KUKA KRL program: sps.sub

&ACCESS RVEO
&REL 86
&COMMENT PLC on control
DEF  SPS ( )
  ;FOLD DECLARATIONS
  ;FOLD BASISTECH DECL
  ;Automatik extern
  DECL STATE_T STAT
  DECL MODUS_T MODE
  ;ENDFOLD (BASISTECH DECL)
  ;FOLD USER DECL
  ; Please insert user defined declarations

  ;ENDFOLD (USER DECL)
  ;ENDFOLD (DECLARATIONS)
  ;FOLD INI
  ;FOLD DEFAULT MSG_T
  $MSG_T={MSG_T: VALID FALSE,RELEASE FALSE,TYP #NOTIFY,MODUL[] " ",KEY[] " ",PARAM_TYP #VALUE,PARAM[] " ",DLG_FORMAT[] " ",ANSWER 0}
  ;ENDFOLD (DEFAULT MSG_T)
  ;FOLD AUTOEXT INIT
  INTERRUPT DECL 91 WHEN $PRO_STATE1==#P_FREE DO RESET_OUT ()
  INTERRUPT ON 91
  $LOOP_MSG[]="                                                            "
  MODE=#SYNC
  $H_POS=$H_POS
  ;Automatik extern
  IF $MODE_OP==#EX THEN
    CWRITE($CMD,STAT,MODE,"RUN /R1/CELL()")
  ENDIF
  ;ENDFOLD (AUTOEXT INIT)
  ;FOLD USER INIT
  ; Please insert user defined initialization commands
      sws_set = true

  ;ENDFOLD (USER INIT)
  ;ENDFOLD (INI)

  LOOP
     WAIT FOR NOT($POWER_FAIL)

    ;FOLD USER PLC

; Run toolchanger code
toolchanger()
; Update FTC data
updatetoolforces()




    ;ENDFOLD (USER PLC)
  ENDLOOP
  ;FOLD ;%{H}
  ;FOLD
END
  ;ENDFOLD


DEF  RESET_OUT ( )
  INT N
  $LOOP_MSG[]="                                                            "
  IF REFLECT_PROG_NR == 1 THEN
    FOR N = 0 TO PGNO_LENGTH - 1
      $OUT[PGNO_FBIT_REFL + N] = FALSE
    ENDFOR
  ENDIF
  IF (PGNO_REQ>0) THEN
    $OUT[PGNO_REQ]=FALSE
  ELSE
    IF (PGNO_REQ<0) THEN
      $OUT[-PGNO_REQ]=TRUE
    ENDIF
  ENDIF
END

;FOLD USER SUBROUTINE
; Integrate your user defined subroutines

;ENDFOLD (USER SUBROUTINE)
;ENDFOLD
